ADAPTER ISludgeBuffer (* Adapter Interface *)
  (* Standard: 61499-1 *)
  (* Version 0.0, 7/4/2026, Schneider Electric *)
  PACKAGE SE.Nereda;
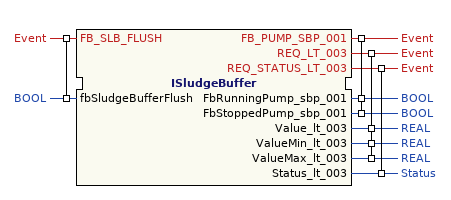
  EVENT_INPUT
    FB_SLB_FLUSH WITH fbSludgeBufferFlush;
  END_EVENT
  EVENT_OUTPUT
    FB_PUMP_SBP_001 WITH FbRunningPump_sbp_001, FbStoppedPump_sbp_001;
    REQ_LT_003 WITH Value_lt_003, ValueMin_lt_003, ValueMax_lt_003;
    REQ_STATUS_LT_003 WITH Status_lt_003;
  END_EVENT
  VAR_INPUT
    fbSludgeBufferFlush : BOOL;
  END_VAR
  VAR_OUTPUT
    FbRunningPump_sbp_001 : BOOL;
    FbStoppedPump_sbp_001 : BOOL;
    Value_lt_003 : REAL;
    ValueMin_lt_003 : REAL;
    ValueMax_lt_003 : REAL;
    Status_lt_003 : Status;
  END_VAR
  SERVICE SOCKET/PLUG
    SEQUENCE request_confirm
      SOCKET.REQ(REQD) -> PLUG.REQ(REQD);
      PLUG.CNF(CNFD) -> SOCKET.CNF(CNFD);
    END_SEQUENCE
    SEQUENCE indication_response
      PLUG.IND(INDD) -> SOCKET.IND(INDD);
      SOCKET.RSP(RSPD) -> PLUG.RSP(RSPD);
    END_SEQUENCE
  END_SERVICE
END_ADAPTER
